TYPE ST_Production_History_DB_Test : // single production data of a station
	STRUCT
		dtStart_time             	: DT ;					// 作業開始時間
		rDuration               	: REAL ;				// unit: sec    (end_time - start_time)
		dtEnd_time               	: DT ;					// 作業結束時間
		usiStation_number         	: USINT ;				// 站點編號
		sStation_name           	: STRING(50) ; 		// 站點名稱
		usiTrack_number           	: USINT ;				// 未定義  Smart Hardcode為1
		usiWpc_number            	: USINT ;				// Shuttle Id
		bPart_ok_overal_results 	: BOOL ;				// 此站點最終判斷/作業結果為OK或NG (彙整站點上的感測器結果及作業結果)
		sSo_number              	: STRING(12) ;			// 由HMI透過ADS告知  (DB中的So資料表需要存在對應資料)
		sFaam_id                	: STRING(20) ;			// 由DB讀取
		diSo_id                  	: DINT ;				// 由HMI透過ADS告知 (DB中的So資料表需要存在對應資料)
	END_STRUCT
END_TYPE

(* stored: Version 1.1.0.1, ProductVersion 3.1.4024.11
   DUT ST_Production_History_DB_Test: Id {734a7360-cf7d-4719-8a64-973399d0e740} *)
